(* PLC project Unnamed, Unknown Unnamed 1 *)
(* stored: creationDateTime 2025-04-12T20:42:18, modificationDateTime 2025-04-18T09:22:19 *)

PROGRAM FLOPS
  VAR
    count AT %MD0 : DINT := 0;
    num_ops AT %MD1 : DINT := 200;
    product AT %MD2 : REAL := 1.0;
    run_flag AT %IX0.0 : BOOL := true;
    reset AT %IX0.1 : BOOL := true;
    run_status AT %QX0.0 : BOOL := false;
  END_VAR
  VAR  (* added by the conversion: wires and edge detectors of the diagram *)
    _MUL2_ENO : BOOL;
    _MUL2_OUT : REAL;
    _SUB7_ENO : BOOL;
    _SUB7_OUT : DINT;
    _GT12_ENO : BOOL;
    _GT12_OUT : BOOL;
    _LE18_ENO : BOOL;
    _LE18_OUT : BOOL;
    _MOVE28_ENO : BOOL;
    _MOVE28_OUT : DINT;
  END_VAR

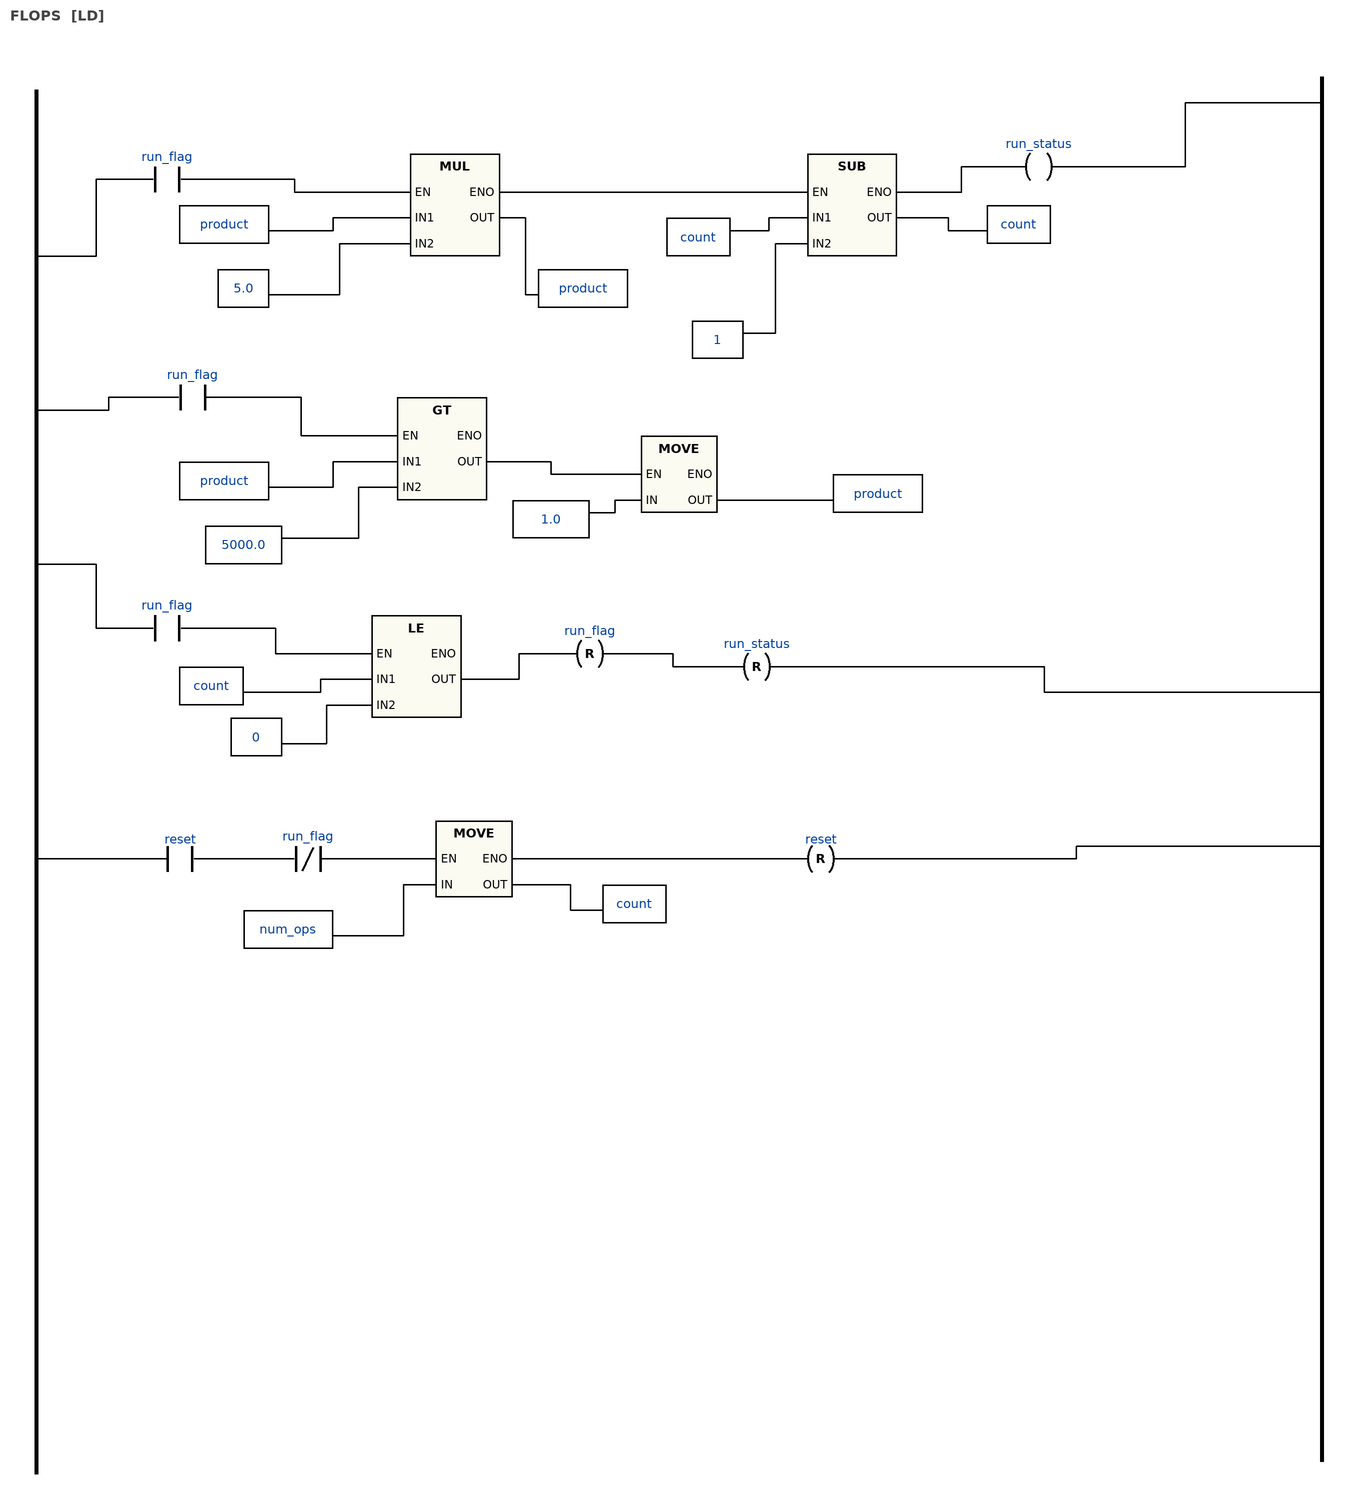
(* LD diagram, written out as Structured Text *)
_MUL2_OUT := MUL(EN := run_flag, IN1 := product, IN2 := 5.0, ENO => _MUL2_ENO);
IF _MUL2_ENO THEN product := _MUL2_OUT; END_IF;
_SUB7_OUT := SUB(EN := _MUL2_ENO, IN1 := count, IN2 := 1, ENO => _SUB7_ENO);
IF _SUB7_ENO THEN count := _SUB7_OUT; END_IF;
_GT12_OUT := GT(EN := run_flag, IN1 := product, IN2 := 5000.0, ENO => _GT12_ENO);
IF _GT12_OUT THEN product := 1.0; END_IF;
_LE18_OUT := LE(EN := run_flag, IN1 := count, IN2 := 0, ENO => _LE18_ENO);
IF _LE18_OUT THEN run_flag := FALSE; END_IF;
_MOVE28_OUT := MOVE(EN := reset AND NOT run_flag, IN := num_ops, ENO => _MOVE28_ENO);
IF _MOVE28_ENO THEN count := _MOVE28_OUT; END_IF;
IF _MOVE28_ENO THEN reset := FALSE; END_IF;
run_status := _SUB7_ENO;
IF _LE18_OUT THEN run_status := FALSE; END_IF;
END_PROGRAM

CONFIGURATION Config0
  RESOURCE Res0 ON PLC
    TASK task0(INTERVAL := T#20ms, PRIORITY := 0);
    PROGRAM instance0 WITH task0 : FLOPS;
  END_RESOURCE
END_CONFIGURATION
